Yaskawa INFORM job: R2_W27-A6(-180,180)_MP_OK.JBI

/JOB
//NAME R2_W27-A6(-180,180)_MP_OK
///FOLDERNAME MP_TEST
//POS
///NPOS 34,34,0,2,0,0
///TOOL 0
///POSTYPE PULSE
///PULSE
C00000=59789,93788,15127,-34295,64393,73036
C00001=119059,-881,-35621,-94148,18883,49989
C00002=83531,-58836,-83505,-107567,-92536,24066
C00003=109115,-94712,-76852,-138223,-101399,5871
C00004=134140,-99016,-76415,-139261,-90415,9289
C00005=134131,-88424,-54946,-139201,-84815,6789
C00006=134127,-86768,-51882,-139151,-84072,6455
C00007=134126,-86092,-50645,-139128,-83774,6321
C00008=134125,-86082,-50640,-139128,-83777,6321
C00009=134126,-86092,-50645,-139128,-83774,6321
C00010=133403,-82234,-43425,-135111,-91400,5238
C00011=133413,-82232,-43424,-135109,-91395,5240
C00012=133403,-82234,-43425,-135111,-91400,5238
C00013=134133,-93654,-65091,-146824,-74524,8479
C00014=134125,-93591,-65063,-146826,-74539,8481
C00015=134124,-92505,-62899,-146704,-73918,8260
C00016=134125,-93591,-65063,-146826,-74539,8481
C00017=133609,-89573,-63522,-146968,-75660,8654
C00018=134131,-93279,-64362,-146784,-74319,8405
C00019=134140,-102529,-84956,-147724,-80724,10608
C00020=84388,-103864,-85424,-146892,-71036,-2051
C00021=126408,-14435,-18329,15377,73761,37506
C00022=131749,-3967,-20197,36380,96853,44141
C00023=134823,3402,-4906,47838,102496,45426
C00024=135841,4647,-106,47495,100367,44867
C00025=136229,5461,2197,47370,99474,44617
C00026=136429,3224,438,47376,99320,44641
C00027=136247,4902,354,47504,100047,44911
C00028=138792,6854,3299,47582,98136,45242
C00029=137845,5671,778,47646,99293,45338
C00030=136838,4359,-4085,47967,101417,45901
C00031=121523,-365,-14274,47607,112143,43536
C00032=116160,-42361,-44579,47879,104974,44952
C00033=65119,-140602,-125961,59810,40226,75337
BC00000=170639,258972,1075158
BC00001=339215,165904,1075165
BC00002=373867,88364,1075171
BC00003=391323,40905,1075175
BC00004=393108,36051,1075175
BC00005=393150,36056,1075175
BC00006=388036,40244,1075175
BC00007=385991,41919,1075175
BC00008=382805,41906,1075175
BC00009=385991,41919,1075175
BC00010=398174,27023,1075175
BC00011=398174,30095,1075175
BC00012=398174,27023,1075175
BC00013=389857,67114,1075175
BC00014=371163,71121,1075175
BC00015=371164,71121,1075175
BC00016=371163,71121,1075175
BC00017=382697,68649,1075175
BC00018=385727,63431,1075175
BC00019=385685,63426,1075175
BC00020=385685,63426,1075175
BC00021=396097,132108,1075175
BC00022=397415,140803,1075175
BC00023=398174,145807,1075175
BC00024=398174,148024,1075175
BC00025=398174,148912,1075175
BC00026=398174,148912,1075175
BC00027=398174,148912,1075175
BC00028=398174,148890,1075175
BC00029=398174,148003,1075175
BC00030=398174,145785,1075175
BC00031=398174,145786,1075171
BC00032=379387,158562,1072617
BC00033=165042,304327,1043479
///POSTYPE BASE
///RECTAN
///RCONF 0,0,0,0,0,0,0,0,0,0,0,0,0,0,0,0,0,0,0,0,0,0,0,0
P00001=2714.263,6838.284,-998.276,27.8833,45.1566,-82.5967
P00006=0.222,-3.123,-1.508,0.0000,0.0000,0.0000
//INST
///DATE 2023/11/16 10:55
///ATTR SC,RW
///GROUP1 RB1,BS1
NOP
'r2_W27-A6(-180,180)
'
'Path S852
SFTOF
MOVJ C00000 BC00000 VJ=20.00
MOVJ C00001 BC00001 VJ=20.00
MOVJ C00002 BC00002 VJ=20.00
MOVJ C00003 BC00003 VJ=20.00
MOVJ C00004 BC00004 VJ=20.00
MOVJ C00005 BC00005 VJ=20.00
MOVL C00006 BC00006 V=100.0
MOVL C00007 BC00007 V=60.0
REFP 3 C00008 BC00008
CALL JOB:SEARCH-R1
SET P001 P006
SFTON P001
MOVL C00009 BC00009 V=60.0
MOVL C00010 BC00010 V=60.0
REFP 3 C00011 BC00011
CALL JOB:SEARCH-R1
SET P001 P006
SFTON P001
MOVL C00012 BC00012 V=60.0
MOVL C00013 BC00013 V=100.0
MOVL C00014 BC00014 V=60.0
REFP 3 C00015 BC00015
CALL JOB:SEARCH-R1
SET P001 P006
SFTON P001
MOVL C00016 BC00016 V=60.0
MOVL C00017 BC00017 V=100.0
MOVL C00018 BC00018 V=100.0
MOVL C00019 BC00019 V=100.0
'Path VIA915
SFTOF
MOVJ C00020 BC00020 VJ=20.00
MOVJ C00021 BC00021 VJ=20.00
MOVJ C00022 BC00022 VJ=20.00
'Path W853
SFTOF
SFTON P001
MOVJ C00023 BC00023 VJ=20.00
MOVL C00024 BC00024 V=100.0
MOVL C00025 BC00025 V=100.0 PL=0
REFP 1 C00026 BC00026
REFP 2 C00027 BC00027
MACRO1 MJ#(0) ARGF7
ARCON
MOVL C00028 BC00028 V=10.8
ARCOF
MOVL C00029 BC00029 V=100.0
MOVL C00030 BC00030 V=100.0
SFTOF
MOVJ C00031 BC00031 VJ=20.00
MOVJ C00032 BC00032 VJ=20.00
MOVJ C00033 BC00033 VJ=20.00
END
